// Mitsubishi GX Works2 project: test_2   PLC: Q03UDV

PROGRAM MAIN
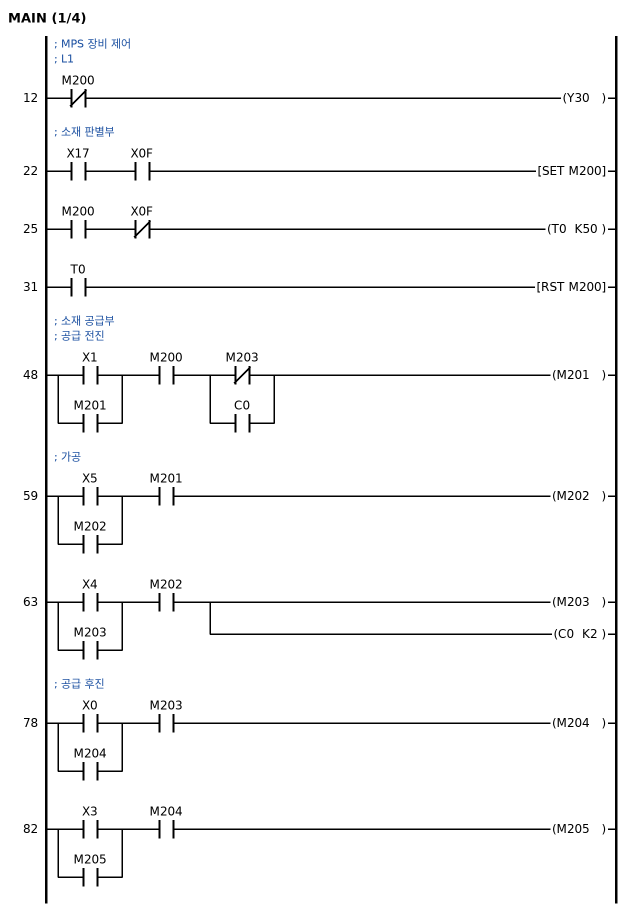
; MPS 장비 제어
; L1
12    LDI     M200
      OUT     Y30
; 소재 판별부
22    LD      X17
      AND     X0F
      SET     M200
25    LD      M200
      ANI     X0F
      OUT     T0 K50
31    LD      T0
      RST     M200
; 소재 공급부
; 공급 전진
48    LD      X1
      OR      M201
      AND     M200
      LDI     M203
      OR      C0
      ANB
      OUT     M201
; 가공
59    LD      X5
      OR      M202
      AND     M201
      OUT     M202
63    LD      X4
      OR      M203
      AND     M202
      OUT     M203
      OUT     C0 K2
; 공급 후진
78    LD      X0
      OR      M204
      AND     M203
      OUT     M204
82    LD      X3
      OR      M205
      AND     M204
      OUT     M205
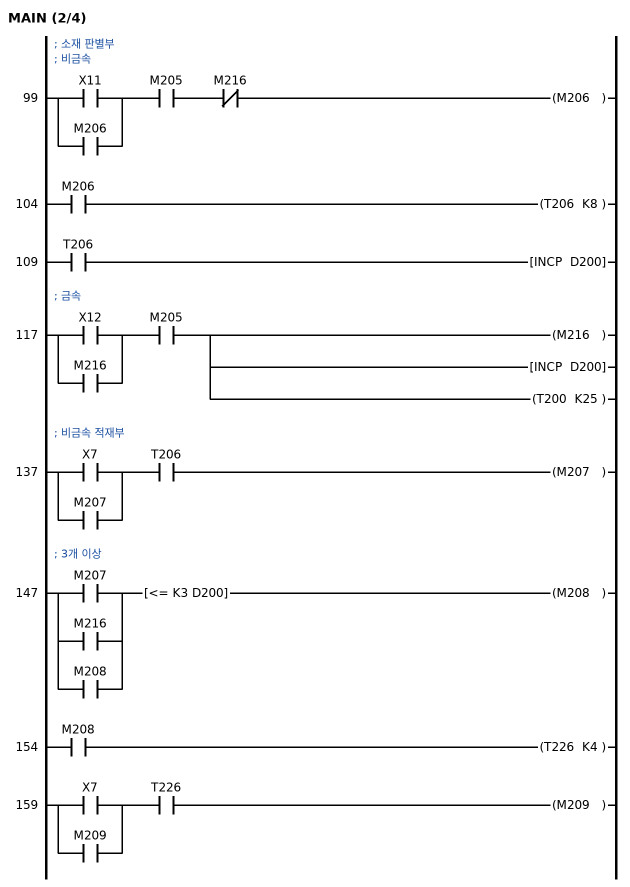
; 소재 판별부
; 비금속
99    LD      X11
      OR      M206
      AND     M205
      ANI     M216
      OUT     M206
104   LD      M206
      OUT     T206 K8
109   LD      T206
      INCP    D200
; 금속
117   LD      X12
      OR      M216
      AND     M205
      OUT     M216
      INCP    D200
      OUT     T200 K25
; 비금속 적재부
137   LD      X7
      OR      M207
      AND     T206
      OUT     M207
; 3개 이상
147   LD      M207
      OR      M216
      OR      M208
      AND<=   K3 D200
      OUT     M208
154   LD      M208
      OUT     T226 K4
159   LD      X7
      OR      M209
      AND     T226
      OUT     M209
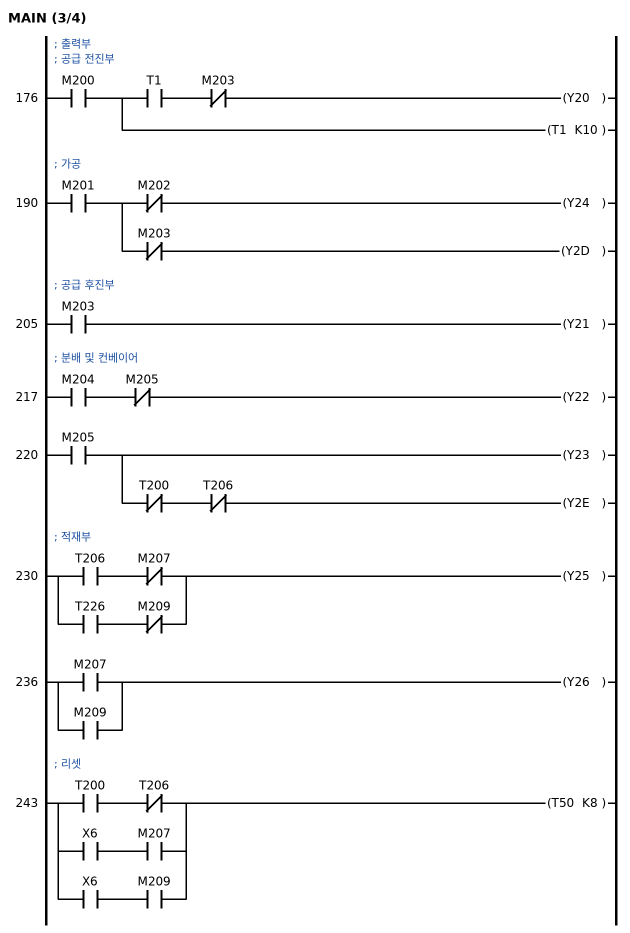
; 출력부
; 공급 전진부
176   LD      M200
      MPS
      AND     T1
      ANI     M203
      OUT     Y20
      MPP
      OUT     T1 K10
; 가공
190   LD      M201
      MPS
      ANI     M202
      OUT     Y24
      MPP
      ANI     M203
      OUT     Y2D
; 공급 후진부
205   LD      M203
      OUT     Y21
; 분배 및 컨베이어
217   LD      M204
      ANI     M205
      OUT     Y22
220   LD      M205
      OUT     Y23
      ANI     T200
      ANI     T206
      OUT     Y2E
; 적재부
230   LD      T206
      ANI     M207
      LD      T226
      ANI     M209
      ORB
      OUT     Y25
236   LD      M207
      OR      M209
      OUT     Y26
; 리셋
243   LD      T200
      ANI     T206
      LD      X6
      AND     M207
      ORB
      LD      X6
      AND     M209
      ORB
      OUT     T50 K8
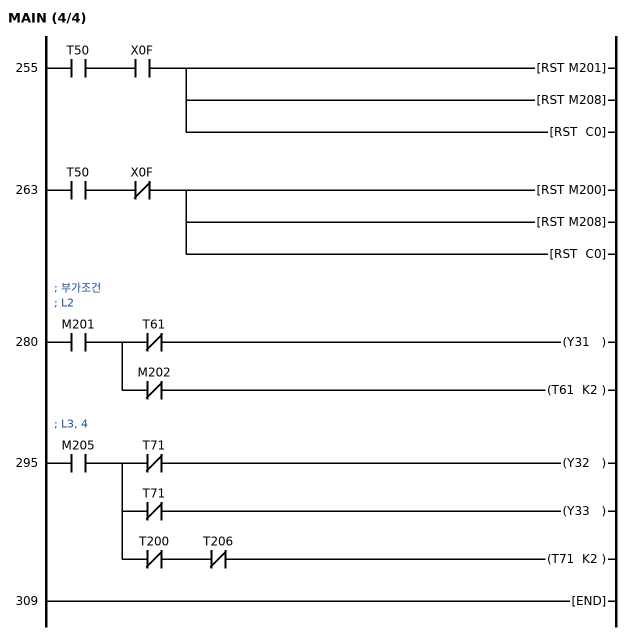
255   LD      T50
      AND     X0F
      RST     M201
      RST     M208
      RST     C0
263   LD      T50
      ANI     X0F
      RST     M200
      RST     M208
      RST     C0
; 부가조건
; L2
280   LD      M201
      MPS
      ANI     T61
      OUT     Y31
      MPP
      ANI     M202
      OUT     T61 K2
; L3, 4
295   LD      M205
      MPS
      ANI     T71
      OUT     Y32
      MRD
      ANI     T71
      OUT     Y33
      MPP
      ANI     T200
      ANI     T206
      OUT     T71 K2
309   END
END_PROGRAM
